{attribute 'OPC.UA.DA.StructuredType' := '1'}
FUNCTION_BLOCK FB_Machine_WaterTreatment_RND EXTENDS FB_BaseMachine IMPLEMENTS I_Machine

VAR_IN_OUT

	{attribute 'OPC.UA.DA' := '0'} 
	stInputs: ST_INPUTS_WaterTreatment_RND;
END_VAR


VAR
	

	bIsFirstRun: BOOL := TRUE;

	
	// Tanks and Sumps
	{attribute 'OPC.UA.DA' := '1'}
  	{attribute 'OPC.UA.DA.StructuredType' := '1'}
	fbTank_CWTA: FB_Tank(TankID:= 'TK1', TankDescr:= 'Clean Water Tank');

	
	{attribute 'OPC.UA.DA' := '1'}
  	{attribute 'OPC.UA.DA.StructuredType' := '1'}
	fbSensor_CWT_A_LSH : FB_Sensor_SICKLevelSwitch_GRF18S(SensorID:= 'TK2A-LSH' , SensorDescr:= 'Clean Water Tank A Level Switch - HIGH', SensorType:= E_SensorType.Analogue);
	
	{attribute 'OPC.UA.DA' := '1'}
  	{attribute 'OPC.UA.DA.StructuredType' := '1'}
	fbUnit_RO_EDI: FB_Unit_RO_RND(UnitID:= 'U1', UnitDescr:= 'Reverse Osmosis (RO) & Electro De-Ionisation (EDI) Unit');
	
	
	// Package all components into structure to pass to sub-FBs 
	// This ST is populated by calling the populateComponents method
	{attribute 'OPC.UA.DA' := '0'} 
	stAllComponents: ST_RNDWTRComponents;
	
	// Interlocks
	{attribute 'OPC.UA.DA' := '1'}
  	{attribute 'OPC.UA.DA.StructuredType' := '1'}
	fbInterlocks: FB_InterlockManager;
	
	
	// Sequence Manager & Sequences
	{attribute 'OPC.UA.DA' := '0'}
	fbSeqWTRMain: FB_SequenceRNDWTR_Main;

	{attribute 'OPC.UA.DA' := '0'}
	aSeqs: ARRAY[1..5] OF FB_SequenceBase;
	
	fbTONStartSequence: TON := (PT := T#10s);
	
END_VAR

fbTONStartSequence();

IF GVL.bAutoUpdateDeviceState THEN
	simulation();       //  <<<----------------- FOR TESTING ONLY, delete this when not being used (it changes devices statet to the target state automatically)
END_IF

IF bIsFirstRun  THEN
	devices_init();	
	sequence_init();
	bIsFirstRun := FALSE;
	fbTONStartSequence(IN := TRUE);
END_IF

IF fbTONStartSequence.Q THEN
	fbSequenceManager.startSequence();
END_IF

scanOPCInputs();
fbSequenceManager(aSequences := aSeqs); //, fbCurrentSequence := aSeqs[1]);
interlocks();


IF GVL.bEnableInterlocks_DM THEN
	interlocks();
END_IF

devices_update();

METHOD checkWaterQuality : BOOL
VAR_INPUT
END_VAR
(*

checkWaterQuality := TRUE;

IF fbSensor_PH.getValue() > stInputs.PH_HIGH_Limit OR 
	fbSensor_PH.getValue() < stInputs.PH_LOW_Limit THEN
	
	checkWaterQuality := FALSE;
	// Raise an event to alert that PH is out of range
END_IF

IF fbSensor_TMP.getValue() > stInputs.Temp_HIGH_Limit OR
	fbSensor_TMP.getValue() < stInputs.Temp_LOW_Limit THEN
	
	checkWaterQuality := FALSE;
	// Raise an event to alert that temp is out of range
END_IF

*)
END_METHOD

METHOD devices_init : BOOL
VAR
	VarInfo : __SYSTEM.VAR_INFO;
END_VAR

fbTank_CWTA.fbSensor_H := fbSensor_CWT_A_LSH;



VarInfo := __VARINFO(fbSensor_CWT_A_LSH );
fbSensor_CWT_A_LSH .setVarID(VarID := VarInfo.Symbol);


VarInfo := __VARINFO(fbUnit_RO_EDI);
fbUnit_RO_EDI.setVarID(VarID := VarInfo.Symbol);



stAllComponents.fbUnit_RO_EDI := ADR( fbUnit_RO_EDI);
// stAllComponents.fbTank_CWTA :=  ADR( fbTank_CWTA);




aAllComponents[1]  :=  ADR(fbUnit_RO_EDI);
//aAllComponents[2]  :=  ADR(fbSensor_CWT_A_LSH );



nQtyComponents := 1;

devices_disable_All();
END_METHOD

METHOD devices_update : BOOL
VAR_INPUT
END_VAR


fbSensor_CWT_A_LSH();
//fbTank_CWTA();
fbUnit_RO_EDI();
END_METHOD

METHOD FB_init : BOOL
VAR_INPUT
	bInitRetains : BOOL; // if TRUE, the retain variables are initialized (warm start / cold start)
	bInCopyCode : BOOL;  // if TRUE, the instance afterwards gets moved into the copy code (online change)


END_VAR
END_METHOD

METHOD interlocks : BOOL
VAR_INPUT
END_VAR
fbInterlocks.init();

fbInterlocks.update(
							Description:= 'RND Clean Water Tank Is Full', 
							InterlockType:= E_InterlockType.RunInterlock, 
							Subject_Device:= ADR(fbUnit_RO_EDI), 
							Subject_State:= E_DeviceState.OFF, 
							Signal:= fbSensor_CWT_A_LSH.getValue() = 0, 
							HoldSequence:= FALSE);
							
fbInterlocks.execute();
END_METHOD

METHOD scanOPCInputs : BOOL
VAR_INPUT
END_VAR

(*
			SEQUENCE CONTROL
*)


IF stInputs.stSequenceManager.Sequence_Ack_Interlock THEN
	fbSequenceManager.acknowledgePause();
	stInputs.stSequenceManager.Sequence_Ack_Interlock := FALSE;
END_IF


CASE stInputs.stSequenceManager.Sequence_Command OF
	E_SequenceState.RUN:
		IF fbSequenceManager.getState() <> E_SequenceState.RUN THEN
			fbSequenceManager.startSequence();
			stInputs.stSequenceManager.Sequence_Command := E_SequenceState.WAIT;
		END_IF
	E_SequenceState.STOP:
		IF fbSequenceManager.getState() <> E_SequenceState.STOP THEN
			fbSequenceManager.stopSequence();
			stInputs.stSequenceManager.Sequence_Command := E_SequenceState.WAIT;
		END_IF
	E_SequenceState.HOLD:
		IF fbSequenceManager.getState() <> E_SequenceState.HOLD THEN
			fbSequenceManager.pauseSequence();
			stInputs.stSequenceManager.Sequence_Command := E_SequenceState.WAIT;
		END_IF
END_CASE
END_METHOD

METHOD sequence_init : BOOL
VAR_INPUT
END_VAR


fbSeqWTRMain(devices := stAllComponents);
fbSeqWTRMain.populateSteps();


aSeqs[1] := fbSeqWTRMain;
END_METHOD

METHOD simulation : BOOL
VAR_INPUT
END_VAR


//fbPump_CleanWaterPumpA.runSimulation();	 
//fbValve_TownWaterSupply.runSimulation();
//fbValve_DM1Supply.runSimulation(); 
//fbUnit_RO_EDI.runSimulation();
END_METHOD

END_FUNCTION_BLOCK

(* stored: Version 1.1.0.1, ProductVersion 3.1.4024.12
   POU FB_Machine_WaterTreatment_RND: Id {91dc64c5-dcc3-4490-9eea-f4a17b38a248}, SpecialFunc None
   Method checkWaterQuality: Id {d1fce34e-1d23-429e-bce0-ac5388c71b7f}
   Method devices_init: Id {b364b7b4-d20f-4c89-9eca-f80ab6e98074}
   Method devices_update: Id {750d125b-cd60-43f0-aa98-578ae4d0bade}
   Method FB_init: Id {78c1d75e-f3cc-43c9-8334-9c51b6a30e07}
   Method interlocks: Id {3d13bd69-2b3a-4c8f-981f-42cbe882feaa}
   Method scanOPCInputs: Id {92f577f2-6ca8-4314-926d-a5f00f73dc03}
   Method sequence_init: Id {63d783dd-7a7b-43fe-b41b-52095ff6a146}
   Method simulation: Id {9f40173e-2ddc-483e-805f-c1b438022de1} *)
